PROGRAM MAIN
VAR
	start : BOOL;
	pingReply : INT := -1; // -1 for not complete, 0 for no ping, 1 for ping reply
	ping : NT_StartProcess;
END_VAR

// you will need to run the following commands on your IPC using Administrator Powershell. 
// this is to install the TcXaeMgmt package in powershell which the below command will use
// ----------------------------------------------------------------------------------------
// [Net.ServicePointManager]::SecurityProtocol = [Net.SecurityProtocolType]::Tls12
// Install-PackageProvider -Name NuGet -MinimumVersion 2.8.5.201 -Force
// Install-Module -Name TcXaeMgmt -RequiredVersion 3.2.25

// To use
// ------
// Main.pingReply is used for the feedback
// 127.0.0.1 is the computer which will be pinged.
// set start to true to run a ping test. 
// typically takes 5 seconds to have a result. 

ping(
	NetId := '',
	PathStr := 'C:\Windows\System32\mshta vbscript:Execute("CreateObject(""WScript.Shell"").Run ""powershell -c $$r=get-adsroute -local;$$s=New-TcSession -Route $$r -Port 851;Write-TcValue -Session $$s -Path ',
	DirName := 'C:\Windows\System32\WindowsPowerShell\v1.0',
	ComndLine := '""""Main.pingReply"""" -value (Test-Connection -ComputerName 127.0.0.1 -Quiet) -Force;Close-TcSession -InputObject $$s;"", 0: window.close")',
	Start := start,
	TmOut := DEFAULT_ADS_TIMEOUT
);

Start := FALSE;

END_PROGRAM

(* stored: Version 1.1.0.1, ProductVersion 3.1.4024.9
   POU MAIN: Id {84c389de-53e5-4ef0-a7de-600428ac4ab5}, SpecialFunc None *)
